FUNCTION_BLOCK FB_NAME IMPLEMENTS I_NAME
VAR_INPUT
END_VAR
VAR_OUTPUT
END_VAR
VAR
	m_name : STRING := 'User';
END_VAR

{warning 'add property implementation'}
PROPERTY Name : STRING
GET
Name := m_name;
END_GET
SET
m_name := Name;
END_SET
END_PROPERTY

{warning 'add method implementation '}
METHOD NUM : INT
NUM := LEN(name);
END_METHOD

END_FUNCTION_BLOCK

(* stored: Version 1.1.0.1, ProductVersion 3.1.4024.3
   POU FB_NAME: Id {1f6171a5-c28c-4620-aa0c-402746ec5b6b}, SpecialFunc None
   Property Name: Id {cdd878a1-1b29-4476-b80d-cb8c3241a4c5}
   Get Get: Id {76212371-b5b0-46e1-9f68-184a9fbf64c8}
   Set Set: Id {a35fa837-806e-4ec2-a2f2-8b6f348d52a6}
   Method NUM: Id {f1cc1750-2061-4ce6-954a-9deeb8f8a44c} *)
